PROGRAM MOTOR2
VAR
END_VAR

io.M2RunControl := io.M2StartSwitch;
io.M2DirectionControl := io.M2DirectionSwitch;
io.M2ConstantControl := io.M2ConstantSwitch;

io.M2RunLight := io.M2RunStatus;
io.M2FaultLight := io.M2FaultStatus;


io.AI1_1 := io.AQ1_1;

END_PROGRAM

(* stored: Version 1.1.0.1, ProductVersion 3.1.4022.12
   POU MOTOR2: Id {32e7a051-6f20-4206-93f6-4507f21fe383}, SpecialFunc None *)
